Staubli VAL3: getSize.pgx

public program getSize(num& x_nSize[])
  local string l_sType
  local string l_sKey
  local num i
  local string l_sItem
  local string l_sPath
begin
  // give back the size to trajectory field
  x_nSize=size(pt:tTraj)
end
